(* Logix 5000 project; controller CLASE_1 Emulate 5570 rev 28.11; software revision 28.02; part 10 of 15 *)
(* tags used below, declared in another part *)
   Inp_PermOK : BOOL;   // 1=Permissives OK, Valve can energize
   Inp_NBPermOK : BOOL;   // 1=Non-Bypassable Permissives OK, valve can energize
   Inp_IntlkOK : BOOL;   // 1=Interlocks OK, valve can energize
   Inp_NBIntlkOK : BOOL;   // 1=Non-Bypassable Interlocks OK, valve can energize
   Inp_IOFault : BOOL;   // Input Communication Status 0=OK, 1=fail
   Inp_Sim : BOOL;   // 1=Simulate working valve; 0=Open/Close/ Monitor actual valve
   Inp_OvrdCmd : DINT;   // Override Mode Command: 0=None, 1=Close, 2=Open
   Inp_Reset : BOOL;   // 1=Reset all fault conditions and latched Alarms
   Cfg_FailOpen : BOOL;   // 1=Fail Open (energize to close), 0=Fail Closed (energize to open)
   Cfg_HasOpenLS : BOOL;   // 1=Valve provides an Open Limit Switch signal
   Cfg_HasClosedLS : BOOL;   // 1=Valve provides a Closed Limit Switch signal
   Cfg_UseOpenLS : BOOL;   // 1=Valve Open LS should be used for failure checking
   Cfg_UseClosedLS : BOOL;   // 1=Valve Closed LS should be used for failure checking
   Cfg_PCmdClear : ALIAS FOR Mode.Cfg_PCmdClear;
   Cfg_OCmdResets : BOOL;   // 1=New Oper valve cmd. resets fault, 0=reset req'd to clear fault
   Cfg_ShedOnFullStall : BOOL;   // 1=Stop Valve and Alarm on Full Stall; 0=Alarm only on Full Stall
   Cfg_ShedOnTransitStall : BOOL;   // 1=Stop Valve and Alarm on Transit Stall; 0=Alarm only on Transit Stall
   Cfg_ShedOnIOFault : BOOL;   // 1=Stop Valve and Alarm on I/O Fault; 0=Alarm only on I/O Fault
   PCmd_Open : BOOL;   // Program Command to Open Valve
   PCmd_Close : BOOL;   // Program Command to Close Valve
   PCmd_Reset : BOOL;   // Program Command to Reset all Alarms requiring Reset
   PCmd_FullStallAck : ALIAS FOR FullStall.PCmd_Ack;   // Program Command to Acknowledge Full Stall Alarm
   PCmd_TransitStallAck : ALIAS FOR TransitStall.PCmd_Ack;   // Program Command to Acknowledge Transit Stall Alarm
   PCmd_IntlkTripAck : ALIAS FOR IntlkTrip.PCmd_Ack;   // Program Command to Acknowledge Interlock Trip Alarm
   PCmd_IOFaultAck : ALIAS FOR IOFault.PCmd_Ack;   // Program Command to Acknowledge I/O Fault Alarm
   OCmd_Open : BOOL;   // Operator Command to Open Valve
   OCmd_Close : BOOL;   // Operator Command to Close Valve
   MCmd_Disable : BOOL;   // Maintenance Command to Disable Valve
   MCmd_Enable : BOOL;   // Maintenance Command to Enable (allow to energize) Valve
   OCmd_Reset : BOOL;   // Operator Command to Reset all Alarms requiring Reset
   OCmd_ResetAckAll : BOOL;   // Operator Command to Reset all Alarms and latched Shed conditions
   Out : BOOL;   // 1=Energize Valve Solenoid
   SrcQ_IO : SINT;   // Source and Quality of primary I/O (enumeration)
   SrcQ : SINT;   // Source and Quality of primary Val/Sts (enumeration)
   Val_Cmd : SINT;   // Device Command 0=None, 1=Close, 2=Open
   Val_Fdbk : SINT;   // Device Feedback 0=Moving, 1=Closed, 2=Opened, 3=Limit Switch Failure
   Val_Sts : SINT;   // Device Confirmed Sts 0=? 1=Closed 2=Open 5=Closing, 6=Opening, 33=Disabled
   Val_Fault : SINT;   // Device Fault Status 0=None, 16=Transit Stall, 17 = Full Stall, 32=I/O Fault, 34=Config Error
   Val_Notify : SINT;   // Current Alarm Level and Acknowledgement (enumeration)
   Sts_Closed : BOOL;   // 1=Valve requested to Close and is confirmed Closed
   Sts_Opening : BOOL;   // 1=Valve requested to open and awaiting open feedback
   Sts_Opened : BOOL;   // 1=Valve requested to open and is confirmed Opened
   Sts_Closing : BOOL;   // 1=Valve requested to Close and awaiting Closed feedback
   Sts_Available : BOOL;   // 1=Valve available for control by automation (Prog)
   Sts_BypActive : BOOL;   // 1=Bypassing Active (Bypassed or Maintenance)
   Sts_Disabled : BOOL;   // 1=Valve is Disabled
   Sts_NotRdy : BOOL;   // 1=Device Not Ready, see detail bits for reason
   Nrdy_Disabled : BOOL;   // 1=Device Not Ready: Device Disabled by Maintenance
   Nrdy_CfgErr : BOOL;   // 1=Device Not Ready: Configuration Error
   Nrdy_Intlk : BOOL;   // 1=Device Not Ready: Interlock Not OK
   Nrdy_Perm : BOOL;   // 1=Device Not Ready: Permissive Not OK
   Nrdy_Fail : BOOL;   // 1=Device Not Ready: Device Failure (Shed Requires Reset)
   Nrdy_IOFault : BOOL;   // 1=Device Not Ready: I/O Fault (Shed Requires Reset)
   Nrdy_NoMode : BOOL;   // 1=Device Not Ready: Device Logic Disabled / NO Mode
   Sts_AlmInh : BOOL;   // 1=An Alarm is Shelved, Disabled or Suppressed, display icon
   Sts_Err : BOOL;   // 1=Error in Config: see detail bits for reason
   Sts_Hand : ALIAS FOR Mode.Sts_Hand;
   Sts_Maint : ALIAS FOR Mode.Sts_Maint;
   Sts_Ovrd : ALIAS FOR Mode.Sts_Ovrd;
   Sts_Prog : ALIAS FOR Mode.Sts_Prog;
   Sts_Oper : ALIAS FOR Mode.Sts_Oper;
   Sts_FullStall : ALIAS FOR FullStall.Inp;   // 1=Valve Full Stall (failed to move at all)
   Sts_TransitStall : ALIAS FOR TransitStall.Inp;   // 1=Valve Transit Stall (did not reach target position)
   Sts_IntlkTrip : ALIAS FOR IntlkTrip.Inp;   // 1=Valve de-energized by an Interlock NOT OK
   Sts_IOFault : ALIAS FOR IOFault.Inp;   // I/O Comm Fault Status (0=OK, 1=Bad)
   Rdy_Open : BOOL;   // 1=Ready to receive OCmd_Open (enables HMI button)
   Rdy_Close : BOOL;   // 1=Ready to receive OCmd_Close (enables HMI button)
   Rdy_Bypass : BOOL;   // 1=Ready to receive OCmd_Bypass (enables HMI button)
   Rdy_Check : BOOL;   // 1=Ready to receive OCmd_Check (enables HMI button)
   Rdy_Disable : BOOL;   // 1=Ready to receive MCmd_Disable (enables HMI button)
   Rdy_Enable : BOOL;   // 1=Ready to receive MCmd_Enable (enables HMI button)
   Rdy_Reset : BOOL;   // 1=Ready to receive OCmd_Reset (enables HMI button)
   Rdy_ResetAckAll : BOOL;   // 1=At least one Alarm or latched Shed condition requires Reset or Ack
   P_ValveSO : BOOL;   // Unique Parameter Name for auto - discovery
   Mode : P_Mode;   // Valve Mode Selection
   IOFault : P_Alarm;   // I/O Fault Alarm
   IntlkTrip : P_Alarm;   // Interlock Trip Alarm
   TransitStall : P_Alarm;   // Valve Transit Stall (moved but did not reach target) Alarm
   FullStall : P_Alarm;   // Valve Full Stall (did not move) Alarm
   Wrk_Open : BOOL;   // 1=Requested to OPEN Valve, 0=Requested to CLOSE Valve
   Wrk_OpenFdbk : BOOL;   // 1=LS Feedback shows valve confirmed open
   Wrk_Notify : DINT;   // Buffer for building Val_Notify
   Wrk_Bypass : BOOL;   // Internal Bypassable Permissives and Interlocks are Bypassed flag
   Wrk_Disabled : BOOL;   // Internal Valve is Disabled
   Wrk_ClosedFdbk : BOOL;   // 1=LS Feedback shows valve confirmed closed
   Wrk_TransitStallT : TIMER;   // Timer for Transit Stall Check
   Wrk_FullStallT : TIMER;   // Timer for Full Stall Check
   Wrk_Cmd : SINT;   // Buffer for building Val_Cmd
   Wrk_Sts : SINT;   // Buffer for building Val_Sts
   Wrk_Fault : SINT;   // Buffer for building Val_Fault
   Wrk_SrcQ : SINT;   // Register for building Source / Quality enumeration
   Wrk_NotRdy : BOOL;   // Device Not Ready conditions excluding shed latches
   Wrk_NoLongerSim : BOOL;   // Switched from Simulated to Real Valve this scan
(* P_ValveSO, continued *)

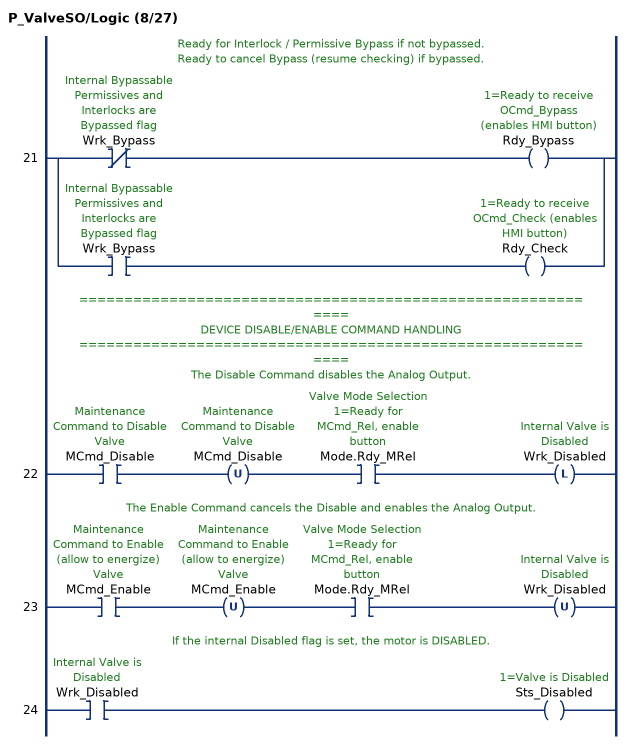
   // Ready for Interlock / Permissive Bypass if not bypassed.
   // Ready to cancel Bypass (resume checking) if bypassed.
   21: [XIO(Wrk_Bypass) OTE(Rdy_Bypass) ,XIC(Wrk_Bypass) OTE(Rdy_Check) ];
   // ============================================================
   // DEVICE DISABLE/ENABLE COMMAND HANDLING
   // ============================================================
   // The Disable Command disables the Analog Output.
   22: XIC(MCmd_Disable)OTU(MCmd_Disable)XIC(Mode.Rdy_MRel)OTL(Wrk_Disabled);
   // The Enable Command cancels the Disable and enables the Analog Output.
   23: XIC(MCmd_Enable)OTU(MCmd_Enable)XIC(Mode.Rdy_MRel)OTU(Wrk_Disabled);
   // If the internal Disabled flag is set, the motor is DISABLED.
   24: XIC(Wrk_Disabled)OTE(Sts_Disabled);
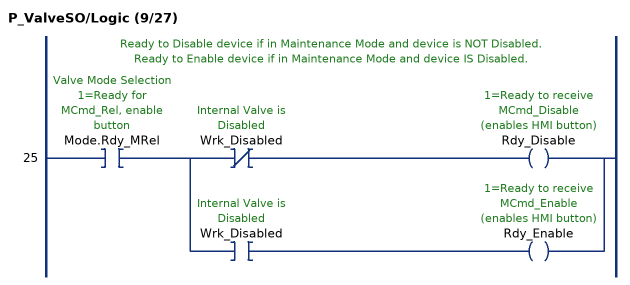
   // Ready to Disable device if in Maintenance Mode and device is NOT Disabled.
   // Ready to Enable device if in Maintenance Mode and device IS Disabled.
   25: XIC(Mode.Rdy_MRel)[XIO(Wrk_Disabled) OTE(Rdy_Disable) ,XIC(Wrk_Disabled) OTE(Rdy_Enable) ];
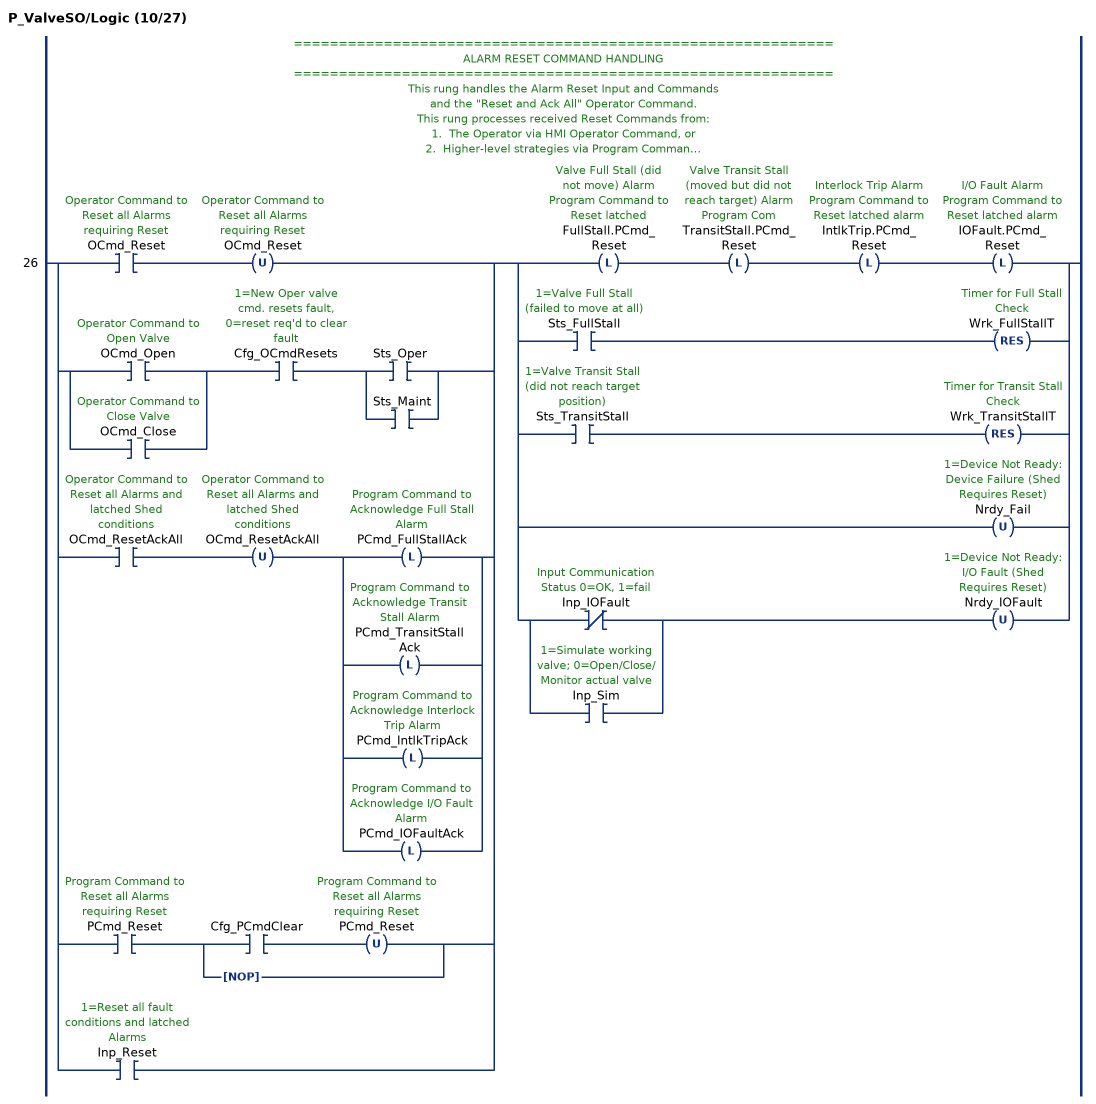
   // ============================================================
   // ALARM RESET COMMAND HANDLING
   // ============================================================
   // This rung handles the Alarm Reset Input and Commands
   // and the "Reset and Ack All" Operator Command.
   // This rung processes received Reset Commands from:
   // 1.  The Operator via HMI Operator Command, or
   // 2.  Higher-level strategies via Program Command
   // 3.  Pushbuttons or other block via Input
   // 4.  Resets initiated by other device Operator Commands (if configured to do so)
   // and forwards the Reset to ALL Alarms and latched Shed conditions.
   // #####  V3.1-00  2014-06-30: Added Not Ready reason bits (Nrdy_xxx)  #####
   // #####  V3.1-01  2014-08-29:  Corrections to Nrdy_ trip and reset logic.  #####
   26: [XIC(OCmd_Reset) OTU(OCmd_Reset) ,[XIC(OCmd_Open) ,XIC(OCmd_Close) ] XIC(Cfg_OCmdResets) [XIC(Sts_Oper) ,XIC(Sts_Maint) ] ,XIC(OCmd_ResetAckAll) OTU(OCmd_ResetAckAll) [OTL(PCmd_FullStallAck) ,OTL(PCmd_TransitStallAck) ,OTL(PCmd_IntlkTripAck) ,OTL(PCmd_IOFaultAck) ] ,XIC(PCmd_Reset) [XIC(Cfg_PCmdClear) OTU(PCmd_Reset) ,NOP() ] ,XIC(Inp_Reset) ][OTL(FullStall.PCmd_Reset) OTL(TransitStall.PCmd_Reset) OTL(IntlkTrip.PCmd_Reset) OTL(IOFault.PCmd_Reset) ,XIC(Sts_FullStall) RES(Wrk_FullStallT) ,XIC(Sts_TransitStall) RES(Wrk_TransitStallT) ,OTU(Nrdy_Fail) ,[XIO(Inp_IOFault) ,XIC(Inp_Sim) ] OTU(Nrdy_IOFault) ];
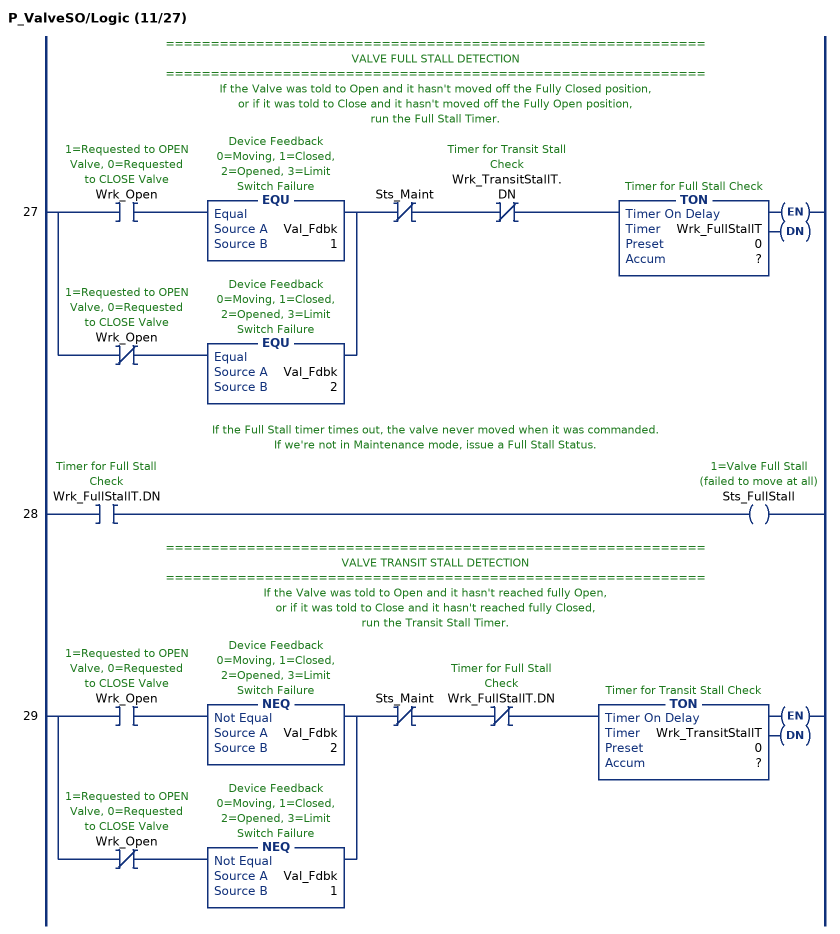
   // ============================================================
   // VALVE FULL STALL DETECTION
   // ============================================================
   // If the Valve was told to Open and it hasn't moved off the Fully Closed position,
   // or if it was told to Close and it hasn't moved off the Fully Open position,
   // run the Full Stall Timer.
   27: [XIC(Wrk_Open) EQU(Val_Fdbk,1) ,XIO(Wrk_Open) EQU(Val_Fdbk,2) ]XIO(Sts_Maint)XIO(Wrk_TransitStallT.DN)TON(Wrk_FullStallT,?,?);
   // If the Full Stall timer times out, the valve never moved when it was commanded.
   // If we're not in Maintenance mode, issue a Full Stall Status.
   28: XIC(Wrk_FullStallT.DN)OTE(Sts_FullStall);
   // ============================================================
   // VALVE TRANSIT STALL DETECTION
   // ============================================================
   // If the Valve was told to Open and it hasn't reached fully Open,
   // or if it was told to Close and it hasn't reached fully Closed,
   // run the Transit Stall Timer.
   29: [XIC(Wrk_Open) NEQ(Val_Fdbk,2) ,XIO(Wrk_Open) NEQ(Val_Fdbk,1) ]XIO(Sts_Maint)XIO(Wrk_FullStallT.DN)TON(Wrk_TransitStallT,?,?);
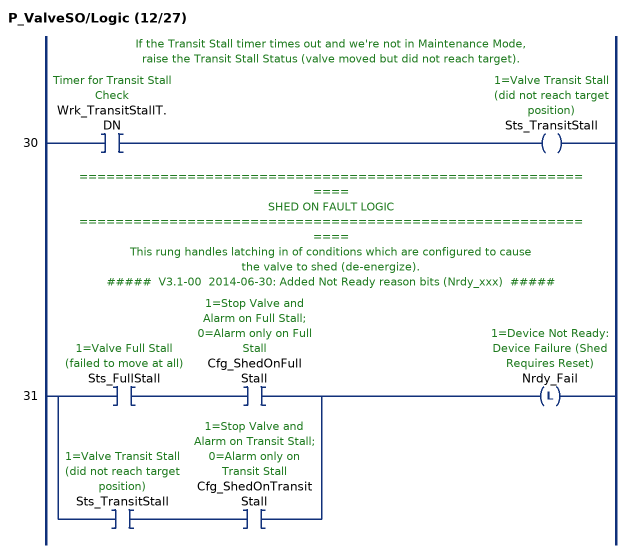
   // If the Transit Stall timer times out and we're not in Maintenance Mode,
   // raise the Transit Stall Status (valve moved but did not reach target).
   30: XIC(Wrk_TransitStallT.DN)OTE(Sts_TransitStall);
   // ============================================================
   // SHED ON FAULT LOGIC
   // ============================================================
   // This rung handles latching in of conditions which are configured to cause
   // the valve to shed (de-energize).
   // #####  V3.1-00  2014-06-30: Added Not Ready reason bits (Nrdy_xxx)  #####
   31: [XIC(Sts_FullStall) XIC(Cfg_ShedOnFullStall) ,XIC(Sts_TransitStall) XIC(Cfg_ShedOnTransitStall) ]OTL(Nrdy_Fail);
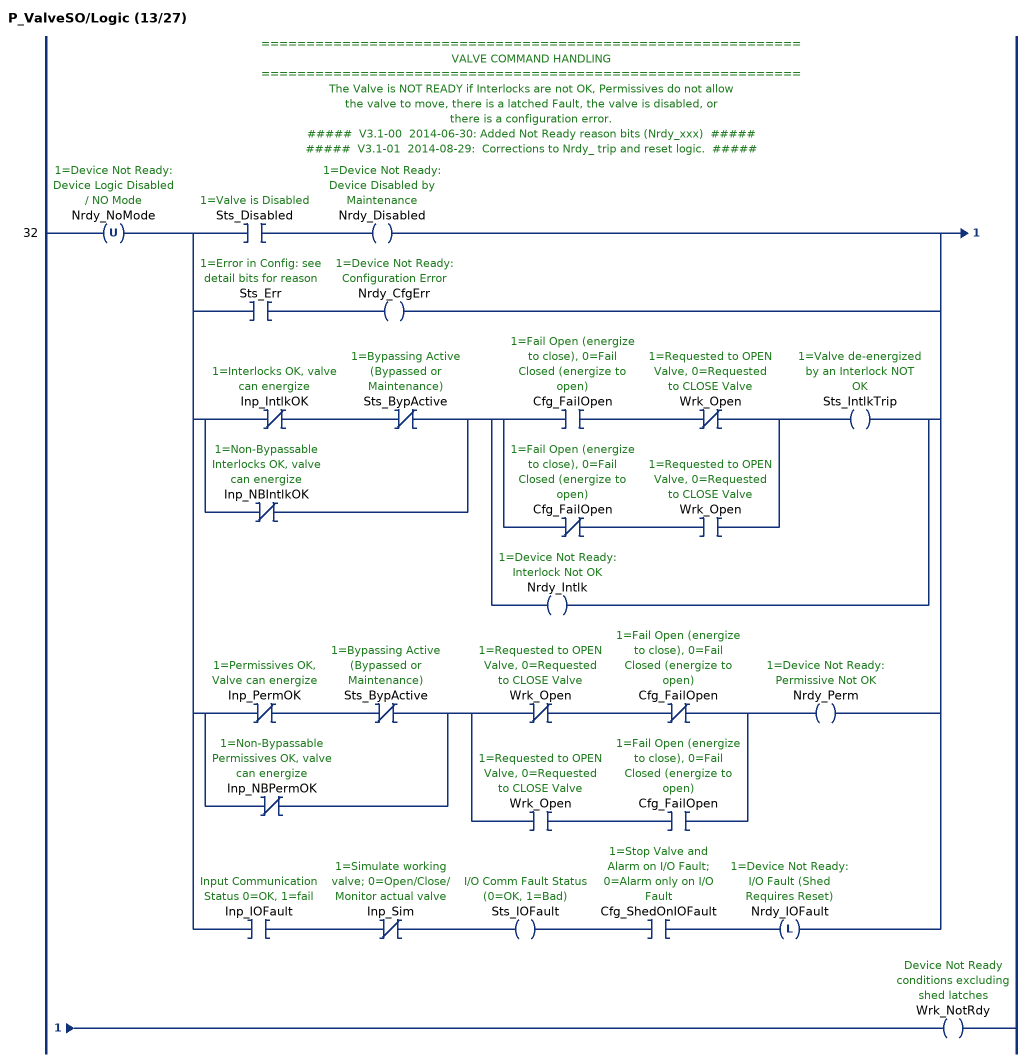
   // ============================================================
   // VALVE COMMAND HANDLING
   // ============================================================
   // The Valve is NOT READY if Interlocks are not OK, Permissives do not allow
   // the valve to move, there is a latched Fault, the valve is disabled, or
   // there is a configuration error.
   // #####  V3.1-00  2014-06-30: Added Not Ready reason bits (Nrdy_xxx)  #####
   // #####  V3.1-01  2014-08-29:  Corrections to Nrdy_ trip and reset logic.  #####
   32: OTU(Nrdy_NoMode)[XIC(Sts_Disabled) OTE(Nrdy_Disabled) ,XIC(Sts_Err) OTE(Nrdy_CfgErr) ,[XIO(Inp_IntlkOK) XIO(Sts_BypActive) ,XIO(Inp_NBIntlkOK) ] [[XIC(Cfg_FailOpen) XIO(Wrk_Open) ,XIO(Cfg_FailOpen) XIC(Wrk_Open) ] OTE(Sts_IntlkTrip) ,OTE(Nrdy_Intlk) ] ,[XIO(Inp_PermOK) XIO(Sts_BypActive) ,XIO(Inp_NBPermOK) ] [XIO(Wrk_Open) XIO(Cfg_FailOpen) ,XIC(Wrk_Open) XIC(Cfg_FailOpen) ] OTE(Nrdy_Perm) ,XIC(Inp_IOFault) XIO(Inp_Sim) OTE(Sts_IOFault) XIC(Cfg_ShedOnIOFault) OTL(Nrdy_IOFault) ]OTE(Wrk_NotRdy);
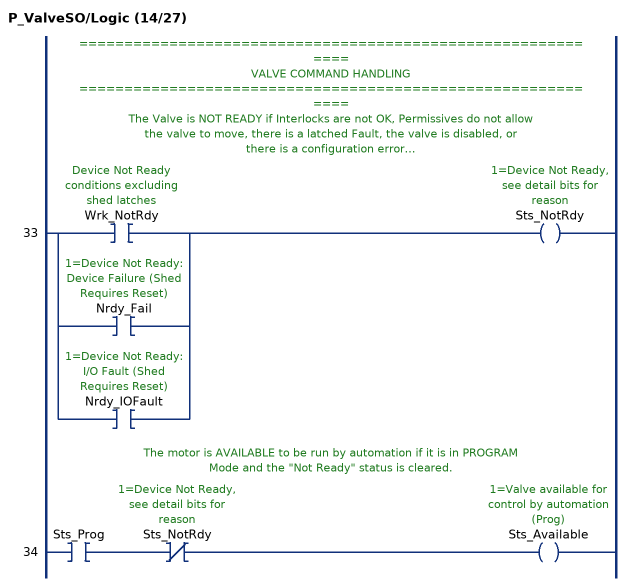
   // ============================================================
   // VALVE COMMAND HANDLING
   // ============================================================
   // The Valve is NOT READY if Interlocks are not OK, Permissives do not allow
   // the valve to move, there is a latched Fault, the valve is disabled, or
   // there is a configuration error.
   // #####  V3.1-00  2014-06-30: Added Not Ready reason bits (Nrdy_xxx)  #####
   // #####  V3.1-01  2014-08-29:  Corrections to Nrdy_ trip and reset logic.  #####
   33: [XIC(Wrk_NotRdy) ,XIC(Nrdy_Fail) ,XIC(Nrdy_IOFault) ]OTE(Sts_NotRdy);
   // The motor is AVAILABLE to be run by automation if it is in PROGRAM
   // Mode and the "Not Ready" status is cleared.
   34: XIC(Sts_Prog)XIO(Sts_NotRdy)OTE(Sts_Available);
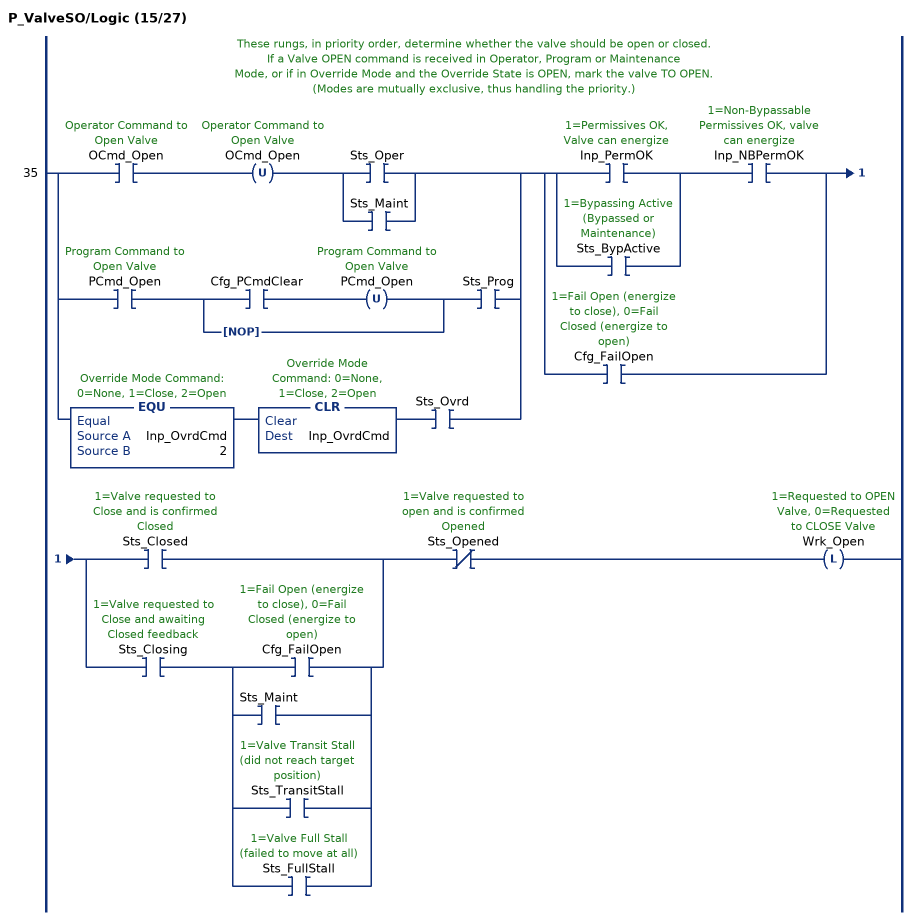
   // These rungs, in priority order, determine whether the valve should be open or closed.
   // If a Valve OPEN command is received in Operator, Program or Maintenance
   // Mode, or if in Override Mode and the Override State is OPEN, mark the valve TO OPEN.
   // (Modes are mutually exclusive, thus handling the priority.)
   35: [XIC(OCmd_Open) OTU(OCmd_Open) [XIC(Sts_Oper) ,XIC(Sts_Maint) ] ,XIC(PCmd_Open) [XIC(Cfg_PCmdClear) OTU(PCmd_Open) ,NOP() ] XIC(Sts_Prog) ,EQU(Inp_OvrdCmd,2) CLR(Inp_OvrdCmd) XIC(Sts_Ovrd) ][[XIC(Inp_PermOK) ,XIC(Sts_BypActive) ] XIC(Inp_NBPermOK) ,XIC(Cfg_FailOpen) ][XIC(Sts_Closed) ,XIC(Sts_Closing) [XIC(Cfg_FailOpen) ,XIC(Sts_Maint) ,XIC(Sts_TransitStall) ,XIC(Sts_FullStall) ] ]XIO(Sts_Opened)OTL(Wrk_Open);
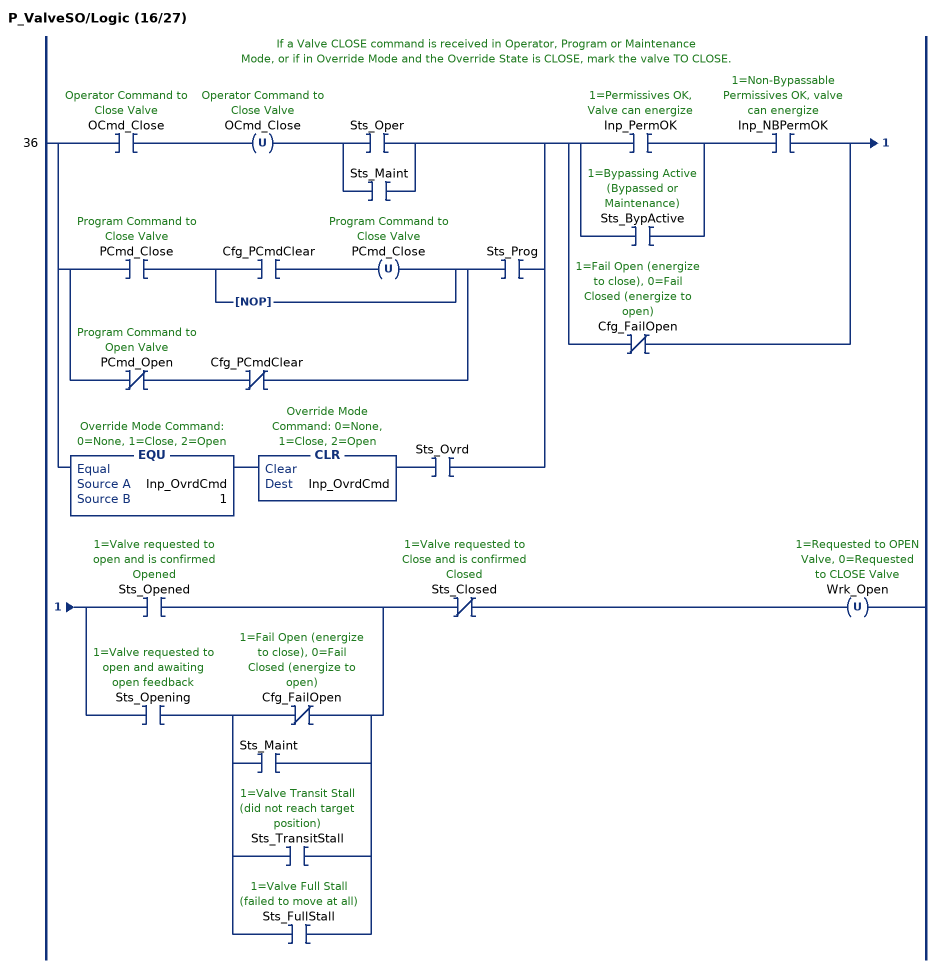
   // If a Valve CLOSE command is received in Operator, Program or Maintenance
   // Mode, or if in Override Mode and the Override State is CLOSE, mark the valve TO CLOSE.
   36: [XIC(OCmd_Close) OTU(OCmd_Close) [XIC(Sts_Oper) ,XIC(Sts_Maint) ] ,[XIC(PCmd_Close) [XIC(Cfg_PCmdClear) OTU(PCmd_Close) ,NOP() ] ,XIO(PCmd_Open) XIO(Cfg_PCmdClear) ] XIC(Sts_Prog) ,EQU(Inp_OvrdCmd,1) CLR(Inp_OvrdCmd) XIC(Sts_Ovrd) ][[XIC(Inp_PermOK) ,XIC(Sts_BypActive) ] XIC(Inp_NBPermOK) ,XIO(Cfg_FailOpen) ][XIC(Sts_Opened) ,XIC(Sts_Opening) [XIO(Cfg_FailOpen) ,XIC(Sts_Maint) ,XIC(Sts_TransitStall) ,XIC(Sts_FullStall) ] ]XIO(Sts_Closed)OTU(Wrk_Open);
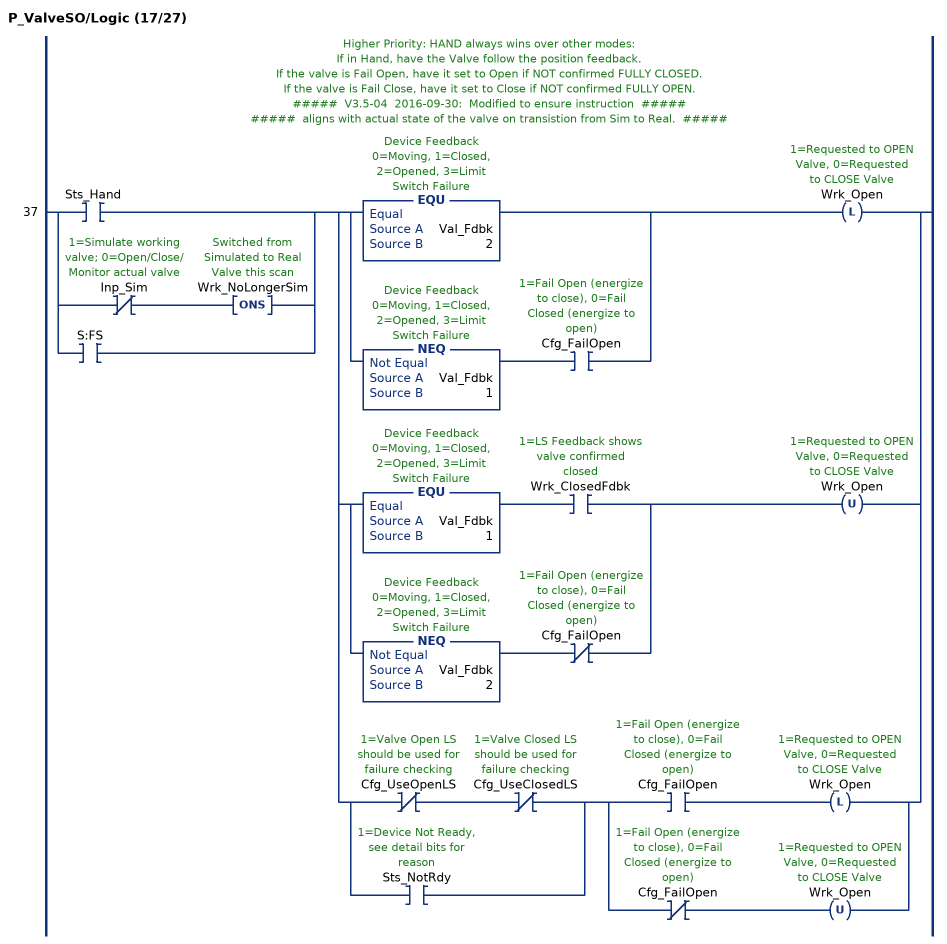
   // Higher Priority: HAND always wins over other modes:
   // If in Hand, have the Valve follow the position feedback.
   // If the valve is Fail Open, have it set to Open if NOT confirmed FULLY CLOSED.
   // If the valve is Fail Close, have it set to Close if NOT confirmed FULLY OPEN.
   // #####  V3.5-04  2016-09-30:  Modified to ensure instruction  #####
   // #####  aligns with actual state of the valve on transistion from Sim to Real.  #####
   37: [XIC(Sts_Hand) ,XIO(Inp_Sim) ONS(Wrk_NoLongerSim) ,XIC(S:FS) ][[EQU(Val_Fdbk,2) ,NEQ(Val_Fdbk,1) XIC(Cfg_FailOpen) ] OTL(Wrk_Open) ,[EQU(Val_Fdbk,1) XIC(Wrk_ClosedFdbk) ,NEQ(Val_Fdbk,2) XIO(Cfg_FailOpen) ] OTU(Wrk_Open) ,[XIO(Cfg_UseOpenLS) XIO(Cfg_UseClosedLS) ,XIC(Sts_NotRdy) ] [XIC(Cfg_FailOpen) OTL(Wrk_Open) ,XIO(Cfg_FailOpen) OTU(Wrk_Open) ] ];
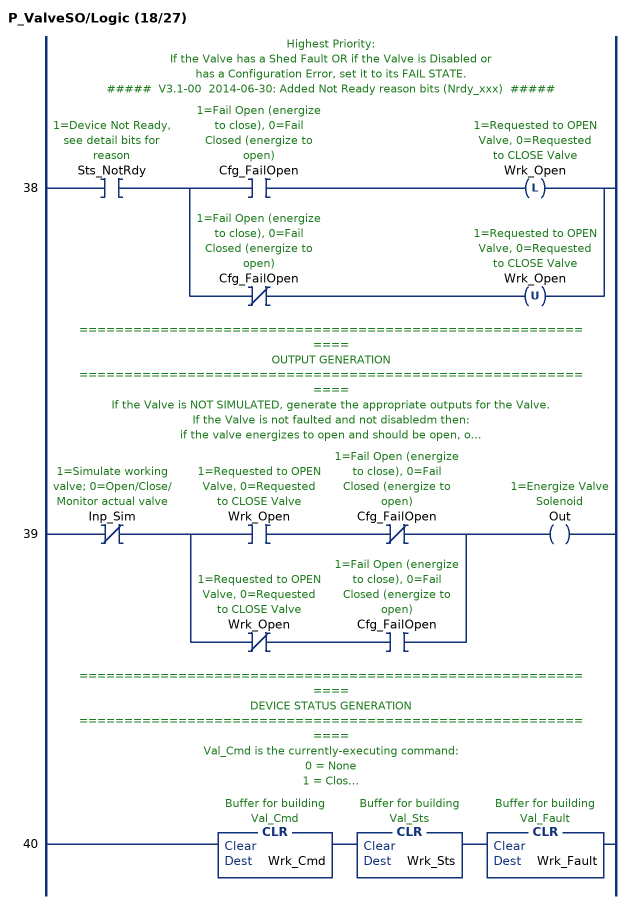
   // Highest Priority:
   // If the Valve has a Shed Fault OR if the Valve is Disabled or
   // has a Configuration Error, set it to its FAIL STATE.
   // #####  V3.1-00  2014-06-30: Added Not Ready reason bits (Nrdy_xxx)  #####
   38: XIC(Sts_NotRdy)[XIC(Cfg_FailOpen) OTL(Wrk_Open) ,XIO(Cfg_FailOpen) OTU(Wrk_Open) ];
   // ============================================================
   // OUTPUT GENERATION
   // ============================================================
   // If the Valve is NOT SIMULATED, generate the appropriate outputs for the Valve.
   // If the Valve is not faulted and not disabledm then:
   // if the valve energizes to open and should be open, or
   // if the valve energizes to close and should be closed,
   // then energize the Output (Out)
   39: XIO(Inp_Sim)[XIC(Wrk_Open) XIO(Cfg_FailOpen) ,XIO(Wrk_Open) XIC(Cfg_FailOpen) ]OTE(Out);
   // ============================================================
   // DEVICE STATUS GENERATION
   // ============================================================
   // Val_Cmd is the currently-executing command:
   // 0 = None
   // 1 = Close
   // 2 = Open
   // Val_Sts is the current device status, as determined by this AOI,
   // based on its knowledge of commands executed and feedback.
   // (This is the status that should be monitored by, for example, FT Historian.)
   // 0 = Powerup / Unknown
   // 1 = Closed
   // 2 = Opened
   // 5 = Closing
   // 6 = Opening
   // 33 = Device Disabled
   // Val_Fault is the current device fault status, as determined by this AOI,
   // based on its knowledge of commands executed and feedback.
   // (This is the fault status that should be monitored by, for example, FT Historian.)
   // 0 = None
   // 16 = Full Stall
   // 17 = Transit Stall
   // 32 = I/O Fault (from Input)
   // 34 = Configuration Error
   40: CLR(Wrk_Cmd)CLR(Wrk_Sts)CLR(Wrk_Fault);
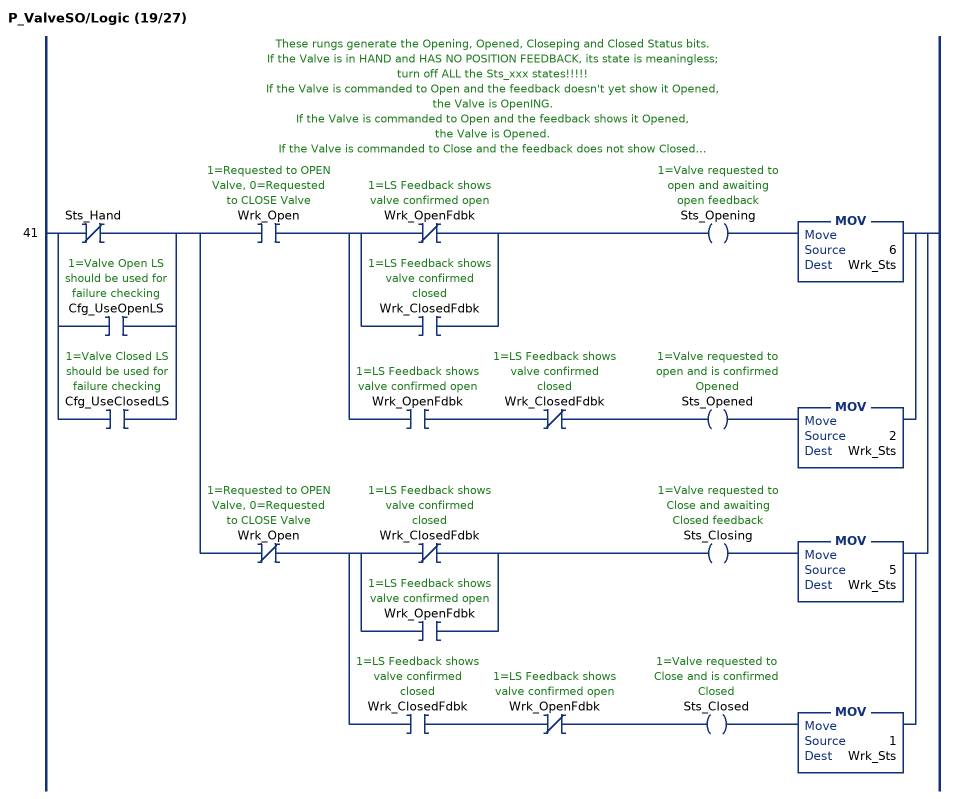
   // These rungs generate the Opening, Opened, Closeping and Closed Status bits.
   // If the Valve is in HAND and HAS NO POSITION FEEDBACK, its state is meaningless;
   // turn off ALL the Sts_xxx states!!!!!
   // If the Valve is commanded to Open and the feedback doesn't yet show it Opened,
   // the Valve is OpenING.
   // If the Valve is commanded to Open and the feedback shows it Opened,
   // the Valve is Opened.
   // If the Valve is commanded to Close and the feedback does not show Closed,
   // the Valve is CloseING.
   // If the Valve is commanded to Close and the feedback shows it has Closed,
   // the Valve is Closed.
   41: [XIO(Sts_Hand) ,XIC(Cfg_UseOpenLS) ,XIC(Cfg_UseClosedLS) ][XIC(Wrk_Open) [[XIO(Wrk_OpenFdbk) ,XIC(Wrk_ClosedFdbk) ] OTE(Sts_Opening) MOV(6,Wrk_Sts) ,XIC(Wrk_OpenFdbk) XIO(Wrk_ClosedFdbk) OTE(Sts_Opened) MOV(2,Wrk_Sts) ] ,XIO(Wrk_Open) [[XIO(Wrk_ClosedFdbk) ,XIC(Wrk_OpenFdbk) ] OTE(Sts_Closing) MOV(5,Wrk_Sts) ,XIC(Wrk_ClosedFdbk) XIO(Wrk_OpenFdbk) OTE(Sts_Closed) MOV(1,Wrk_Sts) ] ];
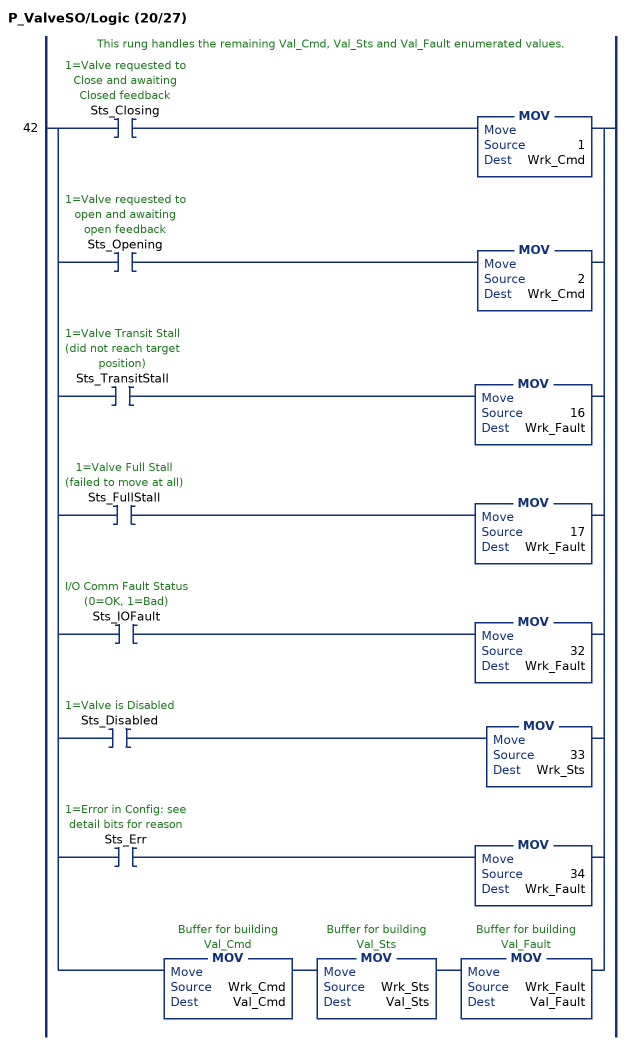
   // This rung handles the remaining Val_Cmd, Val_Sts and Val_Fault enumerated values.
   42: [XIC(Sts_Closing) MOV(1,Wrk_Cmd) ,XIC(Sts_Opening) MOV(2,Wrk_Cmd) ,XIC(Sts_TransitStall) MOV(16,Wrk_Fault) ,XIC(Sts_FullStall) MOV(17,Wrk_Fault) ,XIC(Sts_IOFault) MOV(32,Wrk_Fault) ,XIC(Sts_Disabled) MOV(33,Wrk_Sts) ,XIC(Sts_Err) MOV(34,Wrk_Fault) ,MOV(Wrk_Cmd,Val_Cmd) MOV(Wrk_Sts,Val_Sts) MOV(Wrk_Fault,Val_Fault) ];
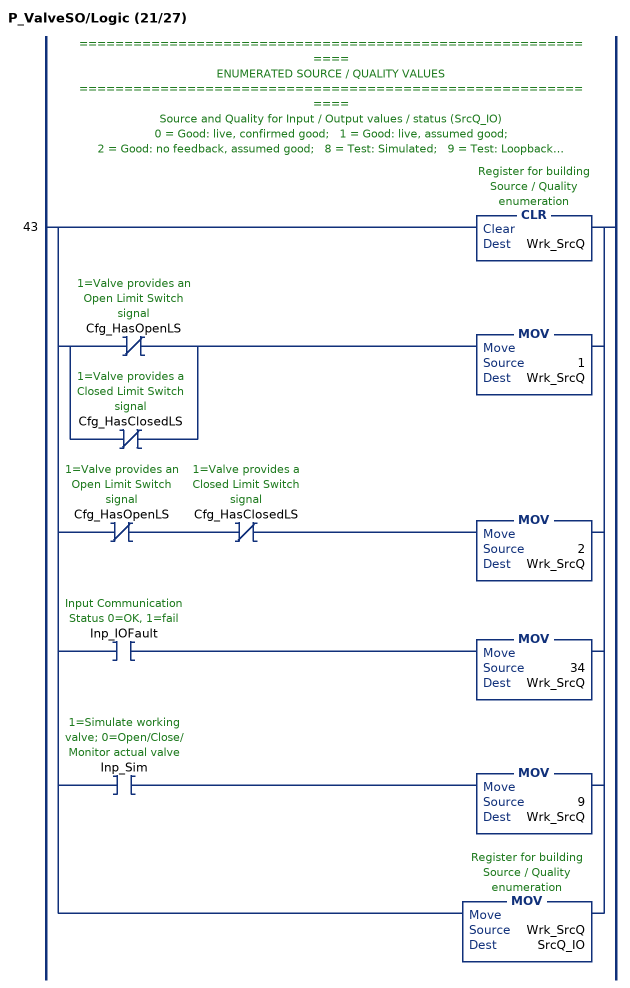
   // ============================================================
   // ENUMERATED SOURCE / QUALITY VALUES
   // ============================================================
   // Source and Quality for Input / Output values / status (SrcQ_IO)
   // 0 = Good: live, confirmed good;   1 = Good: live, assumed good;
   // 2 = Good: no feedback, assumed good;   8 = Test: Simulated;   9 = Test: Loopback;
   // 10 = Test: Manually Entered;   16 = Uncertain: Live, off-spec;
   // 17 = Uncertain, Substituted at Device / Bus;   18 = Uncertain, Substituted at AOI;
   // 19 = Uncertain, using last known good;    20 = Uncertain, using replacement value;
   // 32 = Bad, Signal Failure;   33 = Bad, Channel Fault;
   // 34 = Bad, Module / Comms Fault;   35 = Bad, Invalid Configuration
   // #####  V3.1-00  2014-06-30:  Added rung for Source/Quality enumerations.  #####
   43: [CLR(Wrk_SrcQ) ,[XIO(Cfg_HasOpenLS) ,XIO(Cfg_HasClosedLS) ] MOV(1,Wrk_SrcQ) ,XIO(Cfg_HasOpenLS) XIO(Cfg_HasClosedLS) MOV(2,Wrk_SrcQ) ,XIC(Inp_IOFault) MOV(34,Wrk_SrcQ) ,XIC(Inp_Sim) MOV(9,Wrk_SrcQ) ,MOV(Wrk_SrcQ,SrcQ_IO) ];
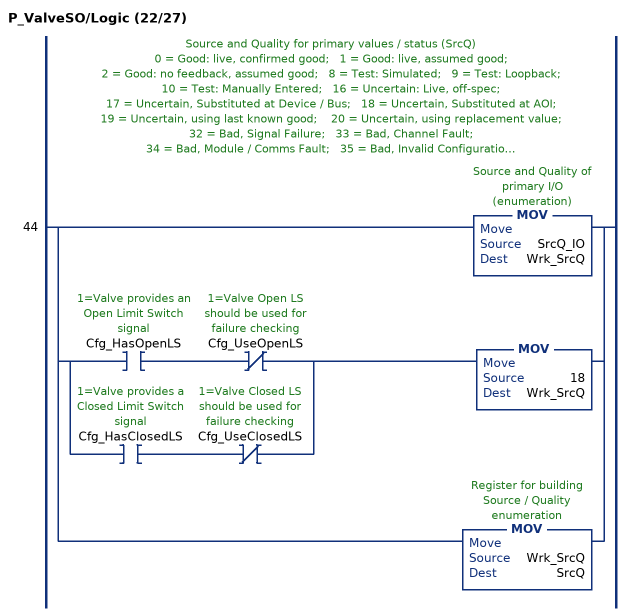
   // Source and Quality for primary values / status (SrcQ)
   // 0 = Good: live, confirmed good;   1 = Good: live, assumed good;
   // 2 = Good: no feedback, assumed good;   8 = Test: Simulated;   9 = Test: Loopback;
   // 10 = Test: Manually Entered;   16 = Uncertain: Live, off-spec;
   // 17 = Uncertain, Substituted at Device / Bus;   18 = Uncertain, Substituted at AOI;
   // 19 = Uncertain, using last known good;    20 = Uncertain, using replacement value;
   // 32 = Bad, Signal Failure;   33 = Bad, Channel Fault;
   // 34 = Bad, Module / Comms Fault;   35 = Bad, Invalid Configuration
   // #####  V3.1-00  2014-06-30:  Added rung for Source/Quality enumerations.  #####
   44: [MOV(SrcQ_IO,Wrk_SrcQ) ,[XIC(Cfg_HasOpenLS) XIO(Cfg_UseOpenLS) ,XIC(Cfg_HasClosedLS) XIO(Cfg_UseClosedLS) ] MOV(18,Wrk_SrcQ) ,MOV(Wrk_SrcQ,SrcQ) ];
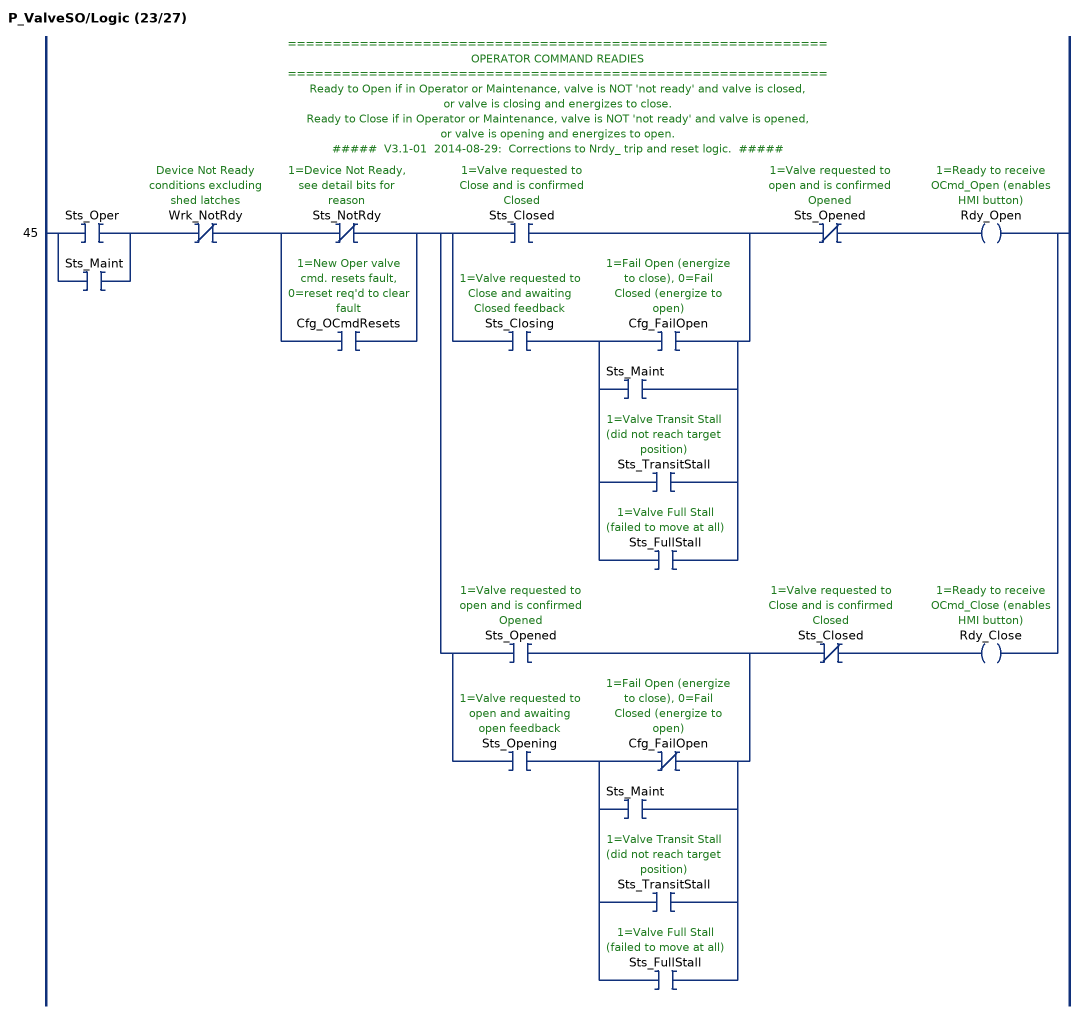
   // ============================================================
   // OPERATOR COMMAND READIES
   // ============================================================
   // Ready to Open if in Operator or Maintenance, valve is NOT 'not ready' and valve is closed,
   // or valve is closing and energizes to close.
   // Ready to Close if in Operator or Maintenance, valve is NOT 'not ready' and valve is opened,
   // or valve is opening and energizes to open.
   // #####  V3.1-01  2014-08-29:  Corrections to Nrdy_ trip and reset logic.  #####
   45: [XIC(Sts_Oper) ,XIC(Sts_Maint) ]XIO(Wrk_NotRdy)[XIO(Sts_NotRdy) ,XIC(Cfg_OCmdResets) ][[XIC(Sts_Closed) ,XIC(Sts_Closing) [XIC(Cfg_FailOpen) ,XIC(Sts_Maint) ,XIC(Sts_TransitStall) ,XIC(Sts_FullStall) ] ] XIO(Sts_Opened) OTE(Rdy_Open) ,[XIC(Sts_Opened) ,XIC(Sts_Opening) [XIO(Cfg_FailOpen) ,XIC(Sts_Maint) ,XIC(Sts_TransitStall) ,XIC(Sts_FullStall) ] ] XIO(Sts_Closed) OTE(Rdy_Close) ];
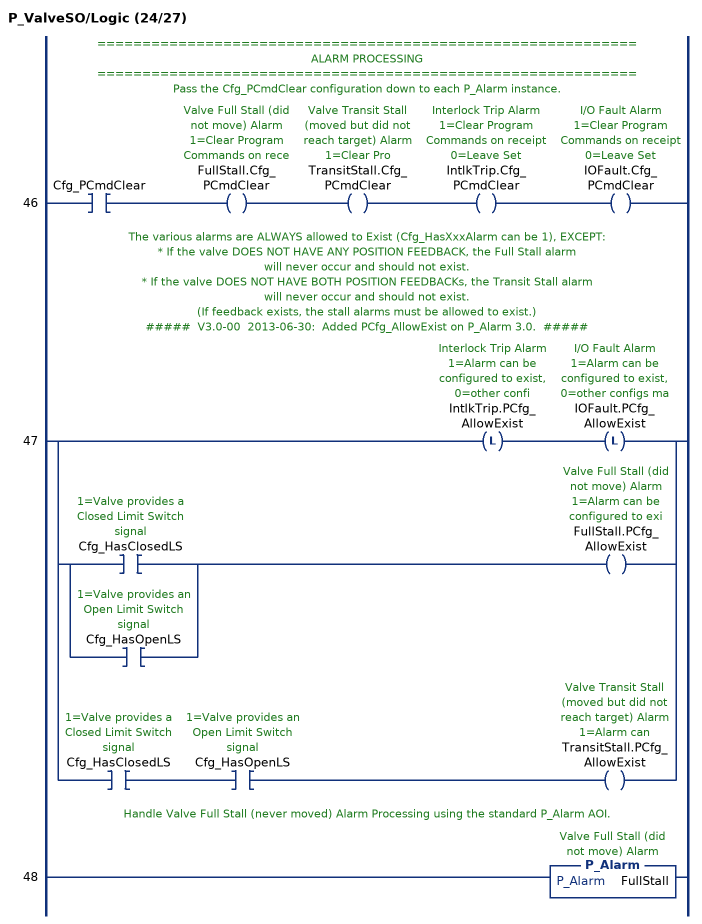
   // ============================================================
   // ALARM PROCESSING
   // ============================================================
   // Pass the Cfg_PCmdClear configuration down to each P_Alarm instance.
   46: XIC(Cfg_PCmdClear)OTE(FullStall.Cfg_PCmdClear)OTE(TransitStall.Cfg_PCmdClear)OTE(IntlkTrip.Cfg_PCmdClear)OTE(IOFault.Cfg_PCmdClear);
   // The various alarms are ALWAYS allowed to Exist (Cfg_HasXxxAlarm can be 1), EXCEPT:
   // * If the valve DOES NOT HAVE ANY POSITION FEEDBACK, the Full Stall alarm
   // will never occur and should not exist.
   // * If the valve DOES NOT HAVE BOTH POSITION FEEDBACKs, the Transit Stall alarm
   // will never occur and should not exist.
   // (If feedback exists, the stall alarms must be allowed to exist.)
   // #####  V3.0-00  2013-06-30:  Added PCfg_AllowExist on P_Alarm 3.0.  #####
   47: [OTL(IntlkTrip.PCfg_AllowExist) OTL(IOFault.PCfg_AllowExist) ,[XIC(Cfg_HasClosedLS) ,XIC(Cfg_HasOpenLS) ] OTE(FullStall.PCfg_AllowExist) ,XIC(Cfg_HasClosedLS) XIC(Cfg_HasOpenLS) OTE(TransitStall.PCfg_AllowExist) ];
   // Handle Valve Full Stall (never moved) Alarm Processing using the standard P_Alarm AOI.
   48: P_Alarm(FullStall);
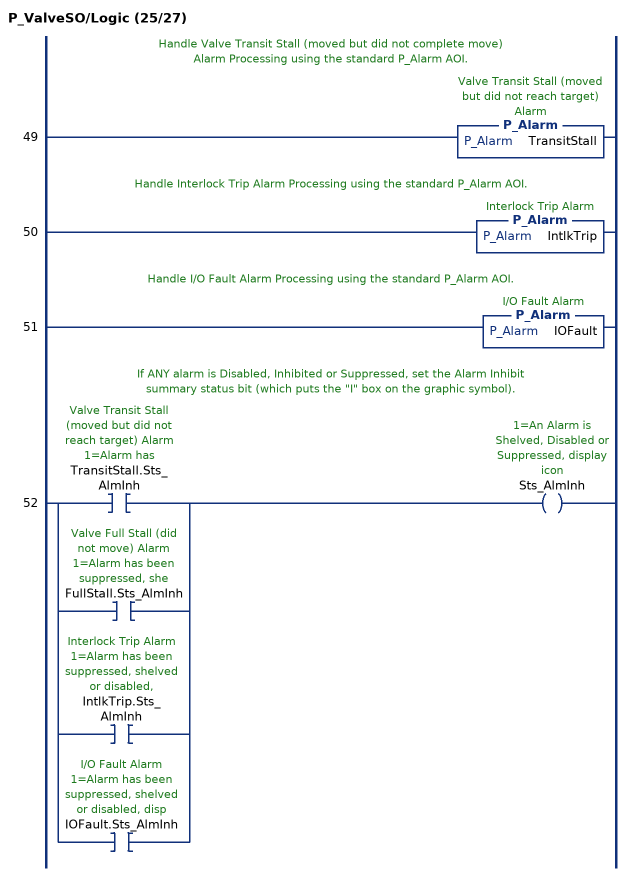
   // Handle Valve Transit Stall (moved but did not complete move)
   // Alarm Processing using the standard P_Alarm AOI.
   49: P_Alarm(TransitStall);
   // Handle Interlock Trip Alarm Processing using the standard P_Alarm AOI.
   50: P_Alarm(IntlkTrip);
   // Handle I/O Fault Alarm Processing using the standard P_Alarm AOI.
   51: P_Alarm(IOFault);
   // If ANY alarm is Disabled, Inhibited or Suppressed, set the Alarm Inhibit
   // summary status bit (which puts the "I" box on the graphic symbol).
   52: [XIC(TransitStall.Sts_AlmInh) ,XIC(FullStall.Sts_AlmInh) ,XIC(IntlkTrip.Sts_AlmInh) ,XIC(IOFault.Sts_AlmInh) ]OTE(Sts_AlmInh);
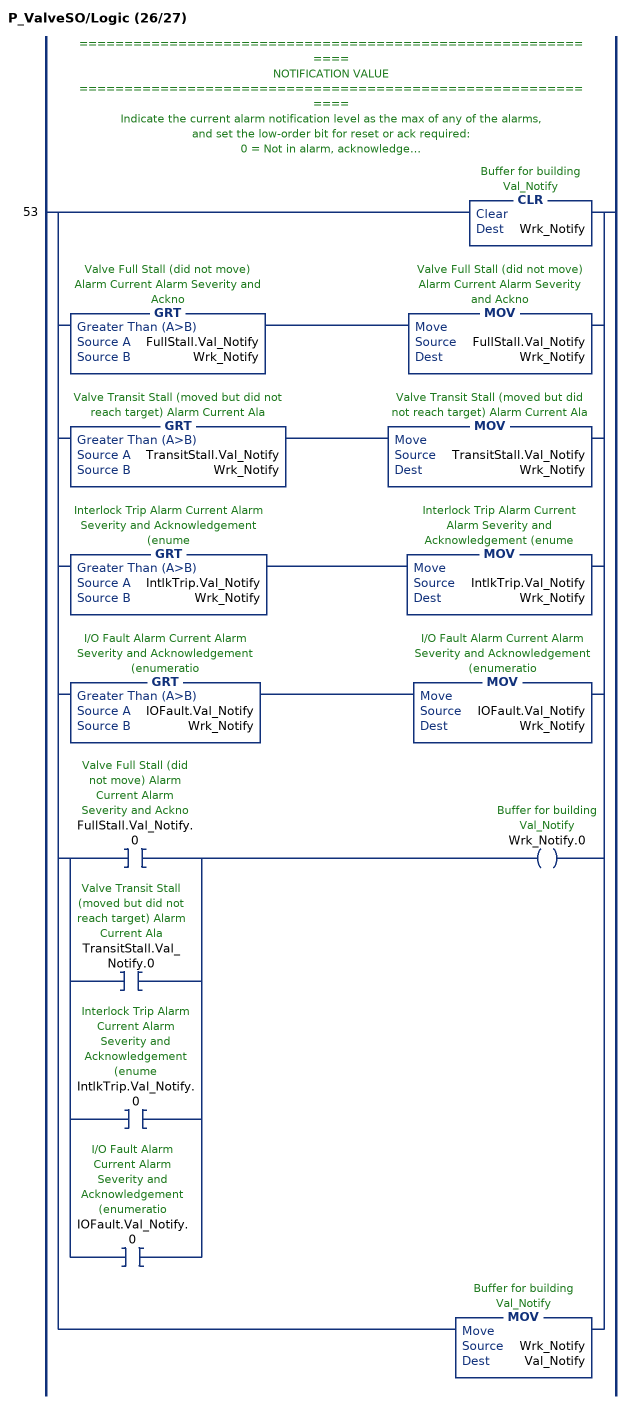
   // ============================================================
   // NOTIFICATION VALUE
   // ============================================================
   // Indicate the current alarm notification level as the max of any of the alarms,
   // and set the low-order bit for reset or ack required:
   // 0 = Not in alarm, acknowledged
   // 1 = Not in alarm, unacknowledged or reset required
   // 2 = Low severity alarm, acknowledged
   // 3 = Low severity alarm, unacknowledged
   // 4 = Medium severity alarm, acknowledged
   // 5 = Medium severity alarm, unacknowledged
   // 6 = High severity alarm, acknowledged
   // 7 = High severity alarm, unacknowledged
   // 8 = Urgent severity alarm, acknowledged
   // 9 = Urgent severity alarm, unacknowledged
   // #####  V3.1-00  2014-06-30:  Separated Reset Reqd functions from Val_Notify  #####
   53: [CLR(Wrk_Notify) ,GRT(FullStall.Val_Notify,Wrk_Notify) MOV(FullStall.Val_Notify,Wrk_Notify) ,GRT(TransitStall.Val_Notify,Wrk_Notify) MOV(TransitStall.Val_Notify,Wrk_Notify) ,GRT(IntlkTrip.Val_Notify,Wrk_Notify) MOV(IntlkTrip.Val_Notify,Wrk_Notify) ,GRT(IOFault.Val_Notify,Wrk_Notify) MOV(IOFault.Val_Notify,Wrk_Notify) ,[XIC(FullStall.Val_Notify.0) ,XIC(TransitStall.Val_Notify.0) ,XIC(IntlkTrip.Val_Notify.0) ,XIC(IOFault.Val_Notify.0) ] OTE(Wrk_Notify.0) ,MOV(Wrk_Notify,Val_Notify) ];
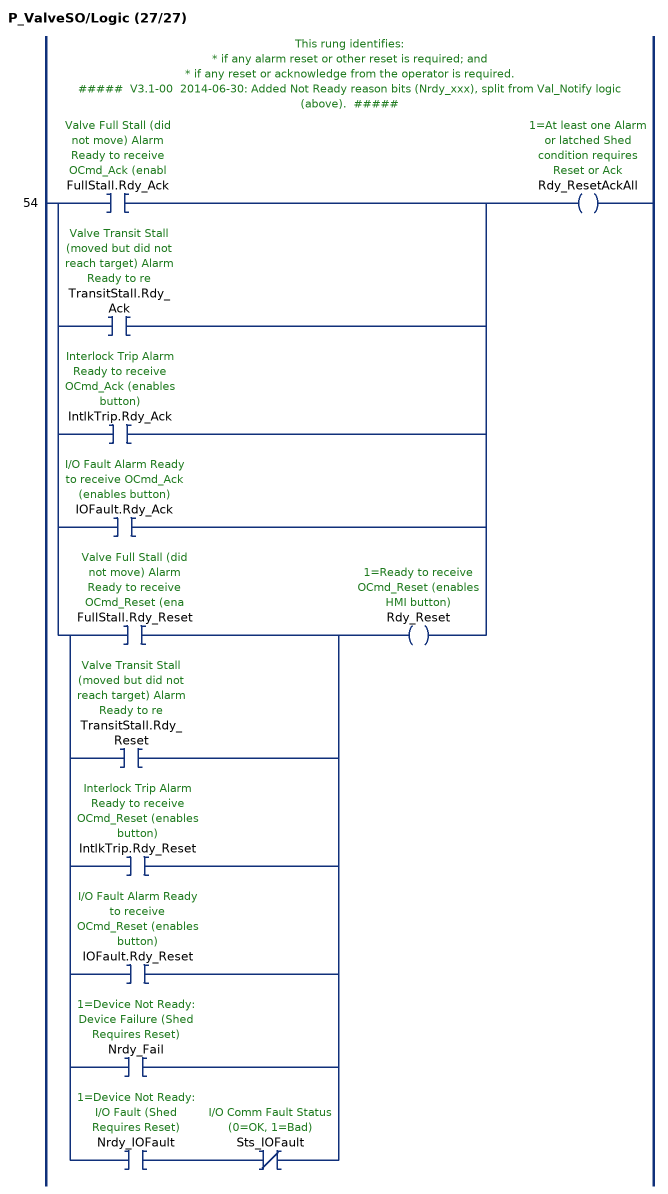
   // This rung identifies:
   // * if any alarm reset or other reset is required; and
   // * if any reset or acknowledge from the operator is required.
   // #####  V3.1-00  2014-06-30: Added Not Ready reason bits (Nrdy_xxx), split from Val_Notify logic (above).  #####
   54: [[XIC(FullStall.Rdy_Ack) ,XIC(TransitStall.Rdy_Ack) ,XIC(IntlkTrip.Rdy_Ack) ,XIC(IOFault.Rdy_Ack) ] ,[XIC(FullStall.Rdy_Reset) ,XIC(TransitStall.Rdy_Reset) ,XIC(IntlkTrip.Rdy_Reset) ,XIC(IOFault.Rdy_Reset) ,XIC(Nrdy_Fail) ,XIC(Nrdy_IOFault) XIO(Sts_IOFault) ] OTE(Rdy_Reset) ]OTE(Rdy_ResetAckAll);
END_ROUTINE
